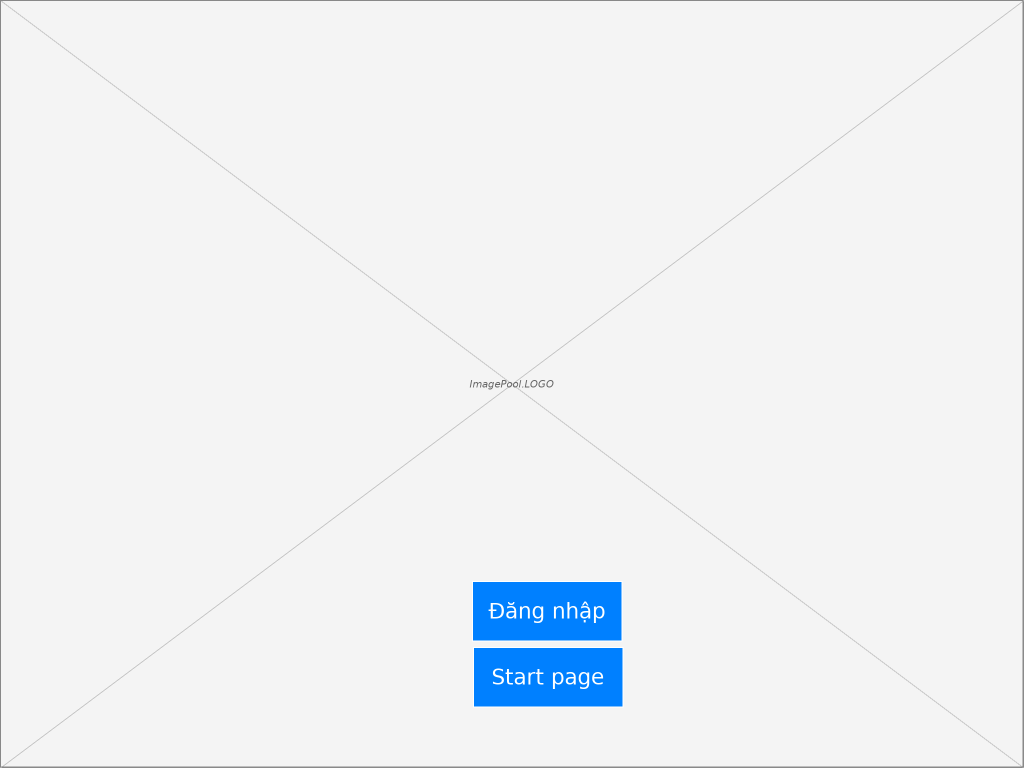
VISUALIZATION N_Login  // 1024x768
    Image (0,0 1024x768), image: ImagePool.LOGO
    Rectangle (472,581 150x60), "Đăng nhập"
        OnMouseDown: VisuUserMgmt Type=Login
    Rectangle (473,647 150x60), "Start page"
        OnMouseDown: execute { username := ''; }
        OnMouseDown: OpenDialog Dialog=startpage, OpenModal=True, OpenCentered=True
END_VISUALIZATION

(* stored: Version 1.1.0.1, ProductVersion 3.1.4024.12
   Visu N_Login: Id {c5642950-31c2-472f-a307-fe1f073a80b1} *)
